(* PLC project PLC, Beckhoff Automation GmbH TwinCAT PLC Control 3.5.20.60 *)
(* stored: creationDateTime 2026-07-21T08:44:36.7013981, modificationDateTime 2026-07-21T08:44:36.7013981 *)

TYPE ST_ADS_API_ScadaViewerApp_PLC_Out_Status_Order :

STRUCT
	
	Valid				:	BOOL;		// |1| Platnost zakázky
	Name				:	STRING;		// |2| Platnost zakázky	
	Count_Expected		:	UINT;		// |3| Očekávaný počet roztříděných mikrospínačů v rámci zakázky
	Count_Actual		:	UINT;		// |4| Aktuální pčoet roztříděných mikrospínačů v rámci zakázky
	
END_STRUCT

END_TYPE
